// TIA Portal project "test4" (V20)

(* hardware
DEVICE "S7-1200 station_1"  S7-1200 Station
   slot 0: "Rack_0"  S7-1200 Rack  Rack  V1.0
   slot 1: "PLC_1"  CPU 1214C DC/DC/DC  6ES7 214-1AG40-0XB0  V4.6
   slot 3: "CB 1241 (RS485)"  CB 1241 (RS485)  6ES7 241-1CH30-1XB0  V1.0
*)

// ===== PLC "PLC_1"  CPU 1214C DC/DC/DC =====

VAR_GLOBAL   // PLC tag table "默认变量表"
   "System_Byte" AT %MB1 : Byte;
   "FirstScan" AT %M1.0 : Bool;
   "DiagStatusUpdate" AT %M1.1 : Bool;
   "AlwaysTRUE" AT %M1.2 : Bool;
   "AlwaysFALSE" AT %M1.3 : Bool;
   "Clock_Byte" AT %MB0 : Byte;
   "Clock_10Hz" AT %M0.0 : Bool;
   "Clock_5Hz" AT %M0.1 : Bool;
   "Clock_2.5Hz" AT %M0.2 : Bool;
   "Clock_2Hz" AT %M0.3 : Bool;
   "Clock_1.25Hz" AT %M0.4 : Bool;
   "Clock_1Hz" AT %M0.5 : Bool;
   "Clock_0.625Hz" AT %M0.6 : Bool;
   "Clock_0.5Hz" AT %M0.7 : Bool;
   "Tag_9" AT %MD1 : Real;
   "Tag_1" AT %MD30 : Real;
   "Tag_10" AT %MD2 : Real;
   "Tag_11" AT %MD31 : Real;
   "Tag_12" AT %MD3 : Real;
   "Tag_13" AT %MD32 : Real;
   "Tag_14" AT %MD4 : Real;
   "Tag_15" AT %MD33 : Real;
   "Tag_16" AT %MD5 : Real;
   "Tag_17" AT %MD34 : Real;
   "Tag_18" AT %MD35 : Real;
   "Tag_19" AT %MD6 : Real;
   "Tag_20" AT %MD7 : Real;
   "Tag_21" AT %MD36 : Real;
   "Tag_22" AT %MD8 : Real;
   "Tag_23" AT %MD37 : Real;
   "Tag_24" AT %MD9 : Real;
   "Tag_25" AT %MD38 : Real;
   "Tag_26" AT %MD10 : Real;
   "Tag_27" AT %MD39 : Real;
   "Tag_28" AT %MD11 : Real;
   "Tag_29" AT %MD40 : Real;
   "Tag_30" AT %MD41 : Real;
   "Tag_31" AT %MD42 : Real;
   "Tag_32" AT %MD12 : Real;
   "Tag_33" AT %MD13 : Real;
END_VAR

DATA_BLOCK "modbusdata1"   // DB3
{ S7_Optimized_Access := 'FALSE' }
VERSION : 0.1
   VAR
      DB1 : Array[0..99] of Int;
   END_VAR
BEGIN
END_DATA_BLOCK

ORGANIZATION_BLOCK "Main"   // OB1, LAD, ProgramCycle
TITLE = "Main Program Sweep (Cycle)"
{ S7_Optimized_Access := 'TRUE' }
VERSION : 0.1
// 使用前必读，该程序基于s7-1200,cpu版本号是v4.6，通讯板是CB1241 RS485的，版本号是V1.0，modbus库是使用V6.0的
   VAR_INPUT
      Initial_Call : Bool;   // Initial call of this OB
      Remanence : Bool;   // =True, if remanent data are available
   END_VAR
BEGIN

REGION Network 1
   // 模块初始化
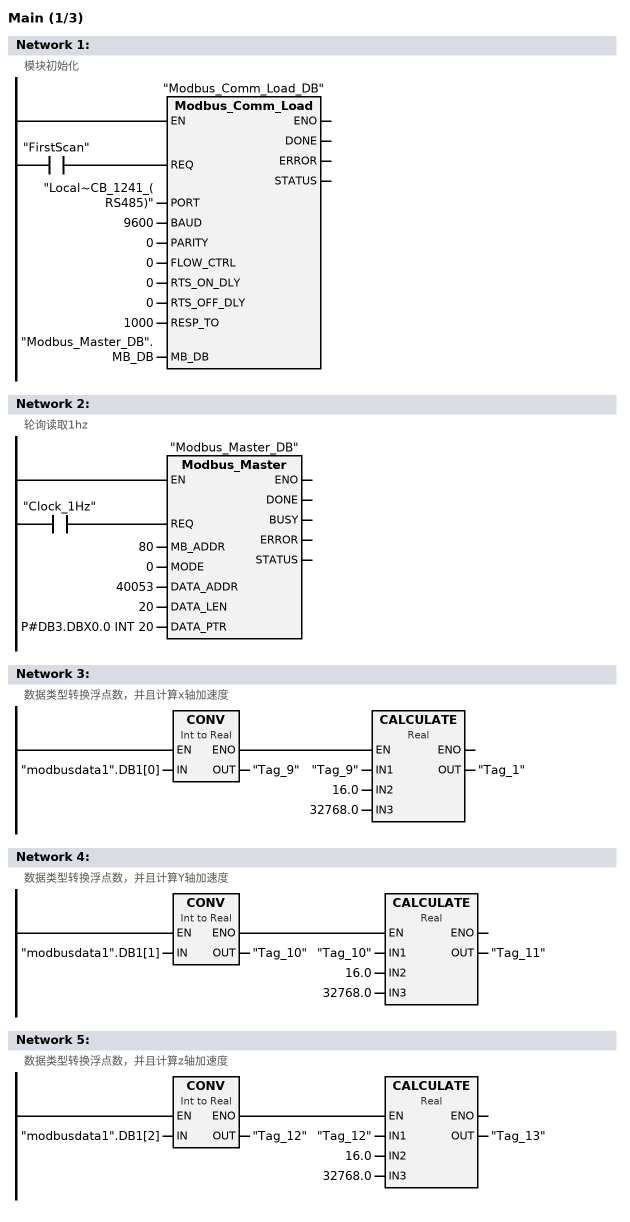
   "Modbus_Comm_Load_DB"(REQ := "FirstScan",   // Modbus_Comm_Load
                         PORT := "Local~CB_1241_(RS485)",
                         BAUD := 9600,
                         PARITY := 0,
                         FLOW_CTRL := 0,
                         RTS_ON_DLY := 0,
                         RTS_OFF_DLY := 0,
                         RESP_TO := 1000,
                         MB_DB := "Modbus_Master_DB".MB_DB);
END_REGION

REGION Network 2
   // 轮询读取1hz
   "Modbus_Master_DB"(REQ := "Clock_1Hz",   // Modbus_Master
                      MB_ADDR := 80,
                      MODE := 0,
                      DATA_ADDR := 40053,
                      DATA_LEN := 20,
                      DATA_PTR := P#DB3.DBX0.0 INT 20);
END_REGION

REGION Network 3
   // 数据类型转换浮点数，并且计算x轴加速度
   RUNG wire#powerrail
      { S7_Templates := "[SrcType := Int, DestType := Real]" } Convert(in := "modbusdata1".DB1[0], out => "Tag_9")
      { S7_Templates := "SrcType := Real"; S7_Expression := "IN1*IN2/IN3" } Calculate(in1 := "Tag_9", in2 := 16.0, in3 := 32768.0, out => "Tag_1")
   END_RUNG
   // the same network as SCL:
   "Tag_9" := INT_TO_REAL("modbusdata1".DB1[0]);
   "Tag_1" := "Tag_9"*16.0/32768.0;
END_REGION

REGION Network 4
   // 数据类型转换浮点数，并且计算Y轴加速度
   RUNG wire#powerrail
      { S7_Templates := "[SrcType := Int, DestType := Real]" } Convert(in := "modbusdata1".DB1[1], out => "Tag_10")
      { S7_Templates := "SrcType := Real"; S7_Expression := "IN1*IN2/IN3" } Calculate(in1 := "Tag_10", in2 := 16.0, in3 := 32768.0, out => "Tag_11")
   END_RUNG
   // the same network as SCL:
   "Tag_10" := INT_TO_REAL("modbusdata1".DB1[1]);
   "Tag_11" := "Tag_10"*16.0/32768.0;
END_REGION

REGION Network 5
   // 数据类型转换浮点数，并且计算z轴加速度
   RUNG wire#powerrail
      { S7_Templates := "[SrcType := Int, DestType := Real]" } Convert(in := "modbusdata1".DB1[2], out => "Tag_12")
      { S7_Templates := "SrcType := Real"; S7_Expression := "IN1*IN2/IN3" } Calculate(in1 := "Tag_12", in2 := 16.0, in3 := 32768.0, out => "Tag_13")
   END_RUNG
   // the same network as SCL:
   "Tag_12" := INT_TO_REAL("modbusdata1".DB1[2]);
   "Tag_13" := "Tag_12"*16.0/32768.0;
END_REGION

REGION Network 6
   // 数据类型转换浮点数，并且计算x轴振动速度
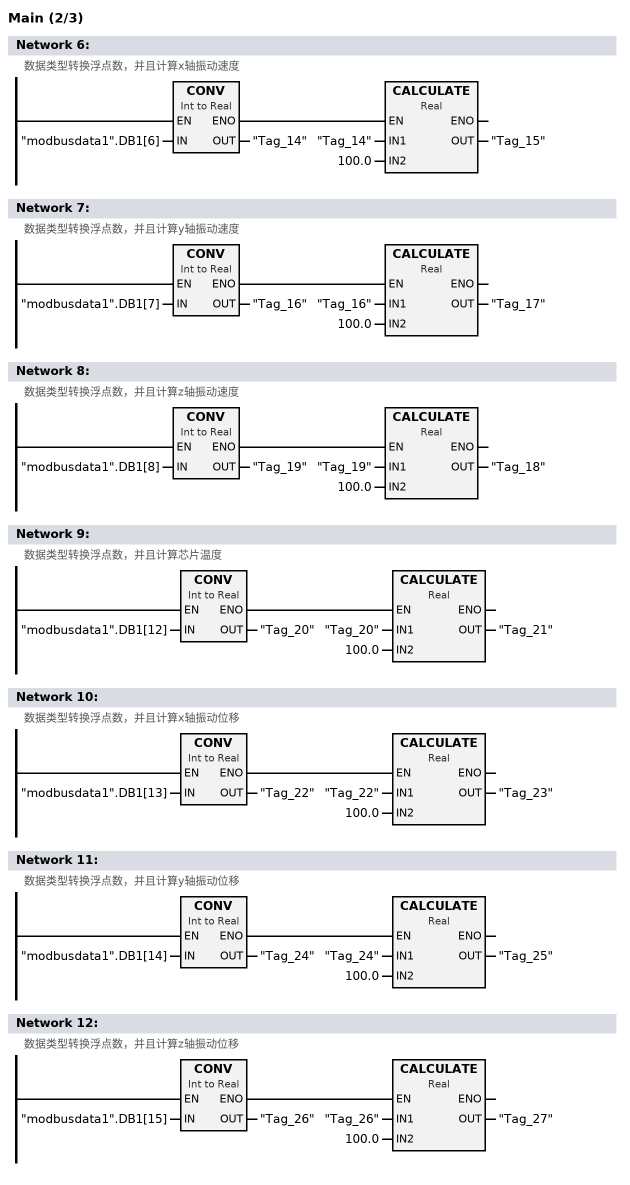
   RUNG wire#powerrail
      { S7_Templates := "[SrcType := Int, DestType := Real]" } Convert(in := "modbusdata1".DB1[6], out => "Tag_14")
      { S7_Templates := "SrcType := Real"; S7_Expression := "IN1/IN2" } Calculate(in1 := "Tag_14", in2 := 100.0, out => "Tag_15")
   END_RUNG
   // the same network as SCL:
   "Tag_14" := INT_TO_REAL("modbusdata1".DB1[6]);
   "Tag_15" := "Tag_14"/100.0;
END_REGION

REGION Network 7
   // 数据类型转换浮点数，并且计算y轴振动速度
   RUNG wire#powerrail
      { S7_Templates := "[SrcType := Int, DestType := Real]" } Convert(in := "modbusdata1".DB1[7], out => "Tag_16")
      { S7_Templates := "SrcType := Real"; S7_Expression := "IN1/IN2" } Calculate(in1 := "Tag_16", in2 := 100.0, out => "Tag_17")
   END_RUNG
   // the same network as SCL:
   "Tag_16" := INT_TO_REAL("modbusdata1".DB1[7]);
   "Tag_17" := "Tag_16"/100.0;
END_REGION

REGION Network 8
   // 数据类型转换浮点数，并且计算z轴振动速度
   RUNG wire#powerrail
      { S7_Templates := "[SrcType := Int, DestType := Real]" } Convert(in := "modbusdata1".DB1[8], out => "Tag_19")
      { S7_Templates := "SrcType := Real"; S7_Expression := "IN1/IN2" } Calculate(in1 := "Tag_19", in2 := 100.0, out => "Tag_18")
   END_RUNG
   // the same network as SCL:
   "Tag_19" := INT_TO_REAL("modbusdata1".DB1[8]);
   "Tag_18" := "Tag_19"/100.0;
END_REGION

REGION Network 9
   // 数据类型转换浮点数，并且计算芯片温度
   RUNG wire#powerrail
      { S7_Templates := "[SrcType := Int, DestType := Real]" } Convert(in := "modbusdata1".DB1[12], out => "Tag_20")
      { S7_Templates := "SrcType := Real"; S7_Expression := "IN1/IN2" } Calculate(in1 := "Tag_20", in2 := 100.0, out => "Tag_21")
   END_RUNG
   // the same network as SCL:
   "Tag_20" := INT_TO_REAL("modbusdata1".DB1[12]);
   "Tag_21" := "Tag_20"/100.0;
END_REGION

REGION Network 10
   // 数据类型转换浮点数，并且计算x轴振动位移
   RUNG wire#powerrail
      { S7_Templates := "[SrcType := Int, DestType := Real]" } Convert(in := "modbusdata1".DB1[13], out => "Tag_22")
      { S7_Templates := "SrcType := Real"; S7_Expression := "IN1/IN2" } Calculate(in1 := "Tag_22", in2 := 100.0, out => "Tag_23")
   END_RUNG
   // the same network as SCL:
   "Tag_22" := INT_TO_REAL("modbusdata1".DB1[13]);
   "Tag_23" := "Tag_22"/100.0;
END_REGION

REGION Network 11
   // 数据类型转换浮点数，并且计算y轴振动位移
   RUNG wire#powerrail
      { S7_Templates := "[SrcType := Int, DestType := Real]" } Convert(in := "modbusdata1".DB1[14], out => "Tag_24")
      { S7_Templates := "SrcType := Real"; S7_Expression := "IN1/IN2" } Calculate(in1 := "Tag_24", in2 := 100.0, out => "Tag_25")
   END_RUNG
   // the same network as SCL:
   "Tag_24" := INT_TO_REAL("modbusdata1".DB1[14]);
   "Tag_25" := "Tag_24"/100.0;
END_REGION

REGION Network 12
   // 数据类型转换浮点数，并且计算z轴振动位移
   RUNG wire#powerrail
      { S7_Templates := "[SrcType := Int, DestType := Real]" } Convert(in := "modbusdata1".DB1[15], out => "Tag_26")
      { S7_Templates := "SrcType := Real"; S7_Expression := "IN1/IN2" } Calculate(in1 := "Tag_26", in2 := 100.0, out => "Tag_27")
   END_RUNG
   // the same network as SCL:
   "Tag_26" := INT_TO_REAL("modbusdata1".DB1[15]);
   "Tag_27" := "Tag_26"/100.0;
END_REGION

REGION Network 13
   // 数据类型转换浮点数，并且计算x轴振动频率
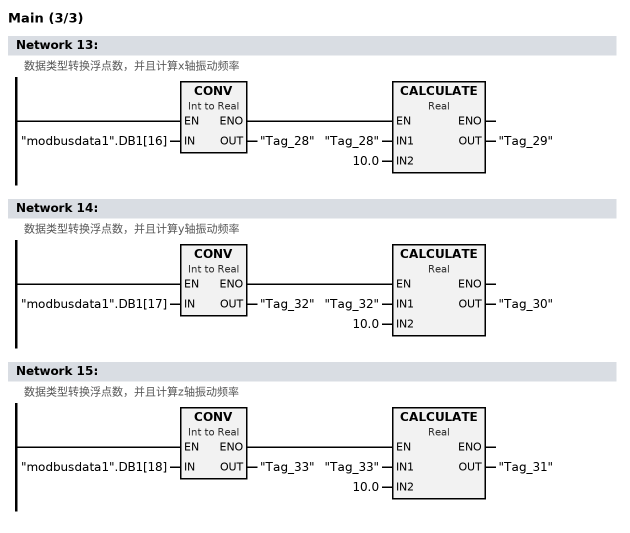
   RUNG wire#powerrail
      { S7_Templates := "[SrcType := Int, DestType := Real]" } Convert(in := "modbusdata1".DB1[16], out => "Tag_28")
      { S7_Templates := "SrcType := Real"; S7_Expression := "IN1/IN2" } Calculate(in1 := "Tag_28", in2 := 10.0, out => "Tag_29")
   END_RUNG
   // the same network as SCL:
   "Tag_28" := INT_TO_REAL("modbusdata1".DB1[16]);
   "Tag_29" := "Tag_28"/10.0;
END_REGION

REGION Network 14
   // 数据类型转换浮点数，并且计算y轴振动频率
   RUNG wire#powerrail
      { S7_Templates := "[SrcType := Int, DestType := Real]" } Convert(in := "modbusdata1".DB1[17], out => "Tag_32")
      { S7_Templates := "SrcType := Real"; S7_Expression := "IN1/IN2" } Calculate(in1 := "Tag_32", in2 := 10.0, out => "Tag_30")
   END_RUNG
   // the same network as SCL:
   "Tag_32" := INT_TO_REAL("modbusdata1".DB1[17]);
   "Tag_30" := "Tag_32"/10.0;
END_REGION

REGION Network 15
   // 数据类型转换浮点数，并且计算z轴振动频率
   RUNG wire#powerrail
      { S7_Templates := "[SrcType := Int, DestType := Real]" } Convert(in := "modbusdata1".DB1[18], out => "Tag_33")
      { S7_Templates := "SrcType := Real"; S7_Expression := "IN1/IN2" } Calculate(in1 := "Tag_33", in2 := 10.0, out => "Tag_31")
   END_RUNG
   // the same network as SCL:
   "Tag_33" := INT_TO_REAL("modbusdata1".DB1[18]);
   "Tag_31" := "Tag_33"/10.0;
END_REGION
END_ORGANIZATION_BLOCK